// Sets the specified number of decimal places for a given real value.
FUNCTION F_SetDecimalPlaces : LREAL // The value with the specified number of decimal places.
VAR_INPUT
	fValue 			: LREAL; // The input floating-point value to be rounded.
	nDecimalPlaces 	: USINT; // The number of decimal places to set the number to.
END_VAR

F_SetDecimalPlaces := EXPT(10, nDecimalPlaces);
F_SetDecimalPlaces := 
	Tc2_Math.LTRUNC(fValue * F_SetDecimalPlaces) / F_SetDecimalPlaces;

END_FUNCTION

(* stored: Version 1.1.0.1
   POU F_SetDecimalPlaces: Id {4c31ee42-2226-0f43-1656-92ad646ccde7}, SpecialFunc None *)
